Universal Robots PolyScope program: programaCubFreedriveStop6-3tcp.urp

Program programaCubFreedriveStop6-3tcp (installation=default directory=/home/ur/ursim-current/programs/provesTFGmireia createdIn=5.15.1 lastSavedIn=5.15.1 robotSerialNumber=20195399999)
Calibrated DH parameters: a=[0, -0.24355, -0.2132, 0, 0, 0]; d=[0.15185, 0, 0, 0.13105, 0.08535, 0.0921]; alpha=[1.570796, 0, 0, 1.570796, -1.570796, 0]; deltaTheta=[0, 0, 0, 0, 0, 0]
InitVariablesNode
Robot Program (runOnlyOnce=true)
  'Definim les variables surtTCP, surtToolFlange i surtMig com a False per indicar quin surt.'
  surtTCP := False
  surtToolFlange := False
  surtMig := False
  'Definim la variable per coneixer la paret que s'esta sortint.'
  valEix := 11
  'Donem valor a la varialbe retrocedir.'
  retrocedir := 0.005
  'Definim els radis de les esferes del TCP, el toolFlange i el punt mig.'
  radiTCP := 0.05
  radiFlange := 0.06
  radiMig := 0.05
  'Agafem els dos punts necessaris per fer un cub perfecte.'
  p1 := p[0.150,-0.483,0.473,0,0,0]
  p2 := p[-0.149,-0.244,0.043,0,0,0]
  'Activem el moviment lliure.'
  Script: freedrive_mode()
  Loop Forever
    'Surt el TCP, el Flange o el punt mig.'
    If surtTCP≟ True  or surtToolFlange≟ True  or surtMig≟ True
      Script: end_freedrive_mode()
      'Eix X positiu es 0 i el negatiu es 10.'
      If valEix≟0
        'ha parat respecte eix X'
        nouPunt := pose_add(get_actual_tcp_pose(), p[-retrocedir,0,0,0,0,0])
        MoveJ speed 20 deg/s, acceleration 30 deg/s^2 (useActiveTCP=true) feature=Base
          Waypoint Variable (Variable): variable=nouPunt
      If valEix≟10
        'ha parat respecte eix X -'
        nouPunt := pose_add(get_actual_tcp_pose(), p[retrocedir,0,0,0,0,0])
        MoveJ speed 20 deg/s, acceleration 30 deg/s^2 (useActiveTCP=true) feature=Base
          Waypoint Variable (Variable): variable=nouPunt
      'Eix Y positiu val 1 i si es el negatiu -1'
      If valEix≟1
        'ha parat respecte eix Y'
        nouPunt := pose_add(get_actual_tcp_pose(), p[0,-retrocedir,0,0,0,0])
        MoveJ speed 20 deg/s, acceleration 30 deg/s^2 (useActiveTCP=true) feature=Base
          Waypoint Variable (Variable): variable=nouPunt
      If valEix≟-1
        'ha parat respecte eix Y -'
        nouPunt := pose_add(get_actual_tcp_pose(), p[0,retrocedir,0,0,0,0])
        MoveJ speed 20 deg/s, acceleration 30 deg/s^2 (useActiveTCP=true) feature=Base
          Waypoint Variable (Variable): variable=nouPunt
      'Eix Z positiu val 2 i si es el negatiu -2 '
      If valEix≟2
        'ha parat respecte eix Z'
        nouPunt := pose_add(get_actual_tcp_pose(), p[0,0,-retrocedir,0,0,0])
        MoveJ speed 20 deg/s, acceleration 30 deg/s^2 (useActiveTCP=true) feature=Base
          Waypoint Variable (Variable): variable=nouPunt
      If valEix≟-2
        'ha parat respecte eix Z -'
        nouPunt := pose_add(get_actual_tcp_pose(), p[0,0,retrocedir,0,0,0])
        MoveJ speed 20 deg/s, acceleration 30 deg/s^2 (useActiveTCP=true) feature=Base
          Waypoint Variable (Variable): variable=nouPunt
      'Retornem les variables a False i reactivem el moviment lliure.'
      surtTCP := False
      surtToolFlange := False
      surtMig := False
      Script: freedrive_mode()
    Wait Sleep waitTime=0.01
Thread Thread_1 (runOnlyOnce=false)
  Loop Forever
    'Obtenim les posicions del TCP, el toolFlange i el punt del mig.'
    llistaPosTCP := get_actual_tcp_pose()
    llistaPosFlange := get_actual_tool_flange_pose()
    llistaPosMig := p[(llistaPosTCP[0]+llistaPosFlange[0])/2,(llistaPosTCP[1]+llistaPosFlange[1])/2,(llistaPosTCP[2]+llistaPosFlange[2])/2,llistaPosTCP[3],llistaPosTCP[4],llistaPosTCP[5]]
    posX := llistaPosTCP[0]
    posXf := llistaPosFlange[0]
    posXm := llistaPosMig[0]
    posY := llistaPosTCP[1]
    posYf := llistaPosFlange[1]
    posYm := llistaPosMig[1]
    posZ := llistaPosTCP[2]
    posZf := llistaPosFlange[2]
    posZm := llistaPosMig[2]
    'Comprovem eixos X'
    If posX≥(p1[0]-radiTCP) or posX≤(p2[0]+radiTCP) (checkContinuously=true)
      surtTCP := True
      If posX≥(p1[0]-radiTCP)
        valEix := 0
      Else 
        valEix := 10
    If posXf≥(p1[0]-radiFlange) or posXf≤(p2[0]+radiFlange) (checkContinuously=true)
      surtToolFlange := True
      If posXf≥(p1[0]-radiFlange)
        valEix := 0
      Else 
        valEix := 10
    If posXm≥(p1[0]-radiMig) or posXm≤(p2[0]+radiMig) (checkContinuously=true)
      surtMig := True
      If posXm≥(p1[0]-radiMig)
        valEix := 0
      Else 
        valEix := 10
    'Comprovem eixos Y'
    If posY≤(p1[1]+radiTCP) or posY≥(p2[1]-radiTCP) (checkContinuously=true)
      surtTCP := True
      If posY≤(p1[1]+radiTCP)
        valEix := -1
      Else 
        valEix := 1
    If posYf≤(p1[1]+radiFlange) or posYf≥(p2[1]-radiFlange) (checkContinuously=true)
      surtToolFlange := True
      If posYf≤(p1[1]+radiFlange)
        valEix := -1
      Else 
        valEix := 1
    If posYm≤(p1[1]+radiMig) or posYm≥(p2[1]-radiMig) (checkContinuously=true)
      surtMig := True
      If posYm≤(p1[1]+radiMig)
        valEix := -1
      Else 
        valEix := 1
    'Comprovem eixos Z'
    If posZ≥(p1[2]-radiTCP) or posZ≤(p2[2]+radiTCP) (checkContinuously=true)
      surtTCP := True
      If posZ≥(p1[2]-radiTCP)
        valEix := 2
      Else 
        valEix := -2
    If posZf≥(p1[2]-radiFlange) or posZf≤(p2[2]+radiFlange) (checkContinuously=true)
      surtToolFlange := True
      If posZf≥(p1[2]-radiFlange)
        valEix := 2
      Else 
        valEix := -2
    If posZm≥(p1[2]-radiMig) or posZm≤(p2[2]+radiMig) (checkContinuously=true)
      surtMig := True
      If posZm≥(p1[2]-radiMig)
        valEix := 2
      Else 
        valEix := -2
